FUNCTION_BLOCK fbTemploopband IMPLEMENTS temp_ITFloopband
VAR_INPUT
END_VAR
VAR_OUTPUT
END_VAR
VAR
	LoopbandActief : BOOL;
	
END_VAR

{warning 'Add method implementation '}
METHOD Beweeg
LoopbandActief:= 1;
END_METHOD

{warning 'Add method implementation '}
METHOD BeweegInLift
END_METHOD

{warning 'Add method implementation '}
METHOD Stop
LoopbandActief:= 0;
END_METHOD

END_FUNCTION_BLOCK

(* stored: Version 1.1.0.1
   POU fbTemploopband: Id {fd55b582-6712-48f5-a30e-f1427c01e92c}, SpecialFunc None
   Method Beweeg: Id {bfbb8d19-dde9-4864-ab11-58c8687d1a19}
   Method BeweegInLift: Id {3e667e89-6b60-4a4e-8b87-7087f7f507b1}
   Method Stop: Id {67bd58cd-8dd1-4983-a51f-8b3ad74bddac} *)
